// TIA Portal project "TIA_Proiect_Sortare_Cutii" (V15.1)

(* hardware
DEVICE "S7-1200 station_1"  S7-1200 Station
   slot 0: "Rack_0"  S7-1200 Rack  Rack  V1.0
   slot 1: "PLC_1"  CPU 1215C DC/DC/Rly  6ES7 215-1HG40-0XB0  V4.1
   slot 2: "DI 8x24VDC_1"  SM 1221 DI8 x 24VDC  6ES7 221-1BF30-0XB0  V1.0
DEVICE "HMI_1"  TP900 Comfort
   slot 0: "HMI_1"  TP900 Comfort  6AV2 124-0JC01-0AX0  15.1.0.0
   slot 1: "HMI_RT_1"  TP900 Comfort  6AV2 124-0JC01-0AX0  15.1.0.0
   slot 5: "HMI_1.IE_CP_1"  PROFINET Interface  15.0.1.0
      slot 1: "PROFINET Interface_1"  PROFINET Interface
         slot 1: "Port_1"  Port
         slot 2: "Port_2"  Port
   slot 7: "HMI_1.MPI/DP_CP_1"  MPI/DP Interface  15.0.1.0
*)

// ===== PLC "PLC_1"  CPU 1215C DC/DC/Rly =====

VAR_GLOBAL   // PLC tag table "Panel"
   "Running" AT %M20.0 : Bool;
   "Panel_IN" AT %I0.0 : "Equip_panel_IN_t";
   "Panel_QD" AT %Q0.0 : "Equip_panel_QD_t";
   "Panel_counter" AT %QW20 : Int;
END_VAR

VAR_GLOBAL   // PLC tag table "BoxLoad_Sorter"
   "BL_entry_sensor" AT %I1.7 : Bool;
   "BL_sorter_IN" AT %I1.0 : "Equip_sorter_IN_t";
   "BL_sorter_QD" AT %Q1.0 : "Equip_sorter_QD_t";
   "BL_entry_conveyor" AT %Q1.4 : Bool;
   "BL_left_conveyor" AT %Q1.5 : Bool;
   "BL_right_conveyor" AT %Q1.6 : Bool;
END_VAR

VAR_GLOBAL   // PLC tag table "Warehouse1"
   "WH1_entry_crane_IN" AT %I2.0 : "Equip_crane_IN_t";
   "WH1_wait_sensor" AT %I2.5 : Bool;
   "WH1_entry_sensor" AT %I2.6 : Bool;
   "WH1_exit_crane_IN" AT %I3.0 : "Equip_crane_IN_t";
   "WH1_exit_sensor" AT %I3.5 : Bool;
   "WH1_entry_crane_QD" AT %Q2.0 : "Equip_crane_QD_t";
   "WH1_entry_crane_TP" AT %QW22 : Int;
   "WH1_exit_crane_TP" AT %QW24 : Int;
   "WH1_exit_crane_QD" AT %Q3.0 : "Equip_crane_QD_t";
   "WH1_load_conveyor" AT %Q2.3 : Bool;
   "WH1_unload_conveyor" AT %Q3.3 : Bool;
   "WH1_exit_conveyor" AT %Q3.4 : Bool;
   "WH1_exit_curved_conveyor" AT %Q3.5 : Bool;
   "WH1_entry_crane_free" AT %M2.0 : Bool;
END_VAR

VAR_GLOBAL   // PLC tag table "Scale1"
   "Elevator1_IN" AT %I4.0 : "Equip_elevator_IN_t";
   "Elevator1_QD" AT %Q4.0 : "Equip_elevator_QD_t";
   "Scale1_entry_sensor" AT %I4.2 : Bool;
   "Scale1_conveyor_sensor" AT %I4.3 : Bool;
   "Elevator1_free" AT %M4.0 : Bool;
END_VAR

VAR_GLOBAL   // PLC tag table "Clock"
   "Clock_10Hz" AT %M0.0 : Bool;
   "Clock_5Hz" AT %M0.1 : Bool;
   "Clock_2.5Hz" AT %M0.2 : Bool;
   "Clock_2Hz" AT %M0.3 : Bool;
   "Clock_1.25Hz" AT %M0.4 : Bool;
   "Clock_1Hz" AT %M0.5 : Bool;
   "Clock_0.625Hz" AT %M0.6 : Bool;
   "Clock_0.5Hz" AT %M0.7 : Bool;
   "Clock_Byte" AT %MB0 : Byte;
END_VAR

TYPE "Info_RFID_t"
   STRUCT
      Serial_Number : Int;
      Box_Type : Int;
      Exit_DateTime : DTL;
   END_STRUCT;
END_TYPE

TYPE "Obj_box_t"
   STRUCT
      Number : Int;
      "Type" : Int;   // 1 - Small box, 2 - Medium box, 3 - Big box
      Weight : Real;
      State : Int;
   END_STRUCT;
END_TYPE

TYPE "Info_OnTime_t"
   STRUCT
      On_time_secs : Int;
      On_time_mins : Int;
      On_time_hours : Int;
   END_STRUCT;
END_TYPE

TYPE "Equip_RFID_t"
   STRUCT
      IN : Struct
         CommandID : Int;
         Status : Int;
         Read_data : Int;
      END_STRUCT;
      QD : Struct
         Command : Int;
         Execute_command : Bool;
         Memory_index : Int;
         Write_data : Int;
      END_STRUCT;
   END_STRUCT;
END_TYPE

// folder: Crane_t

TYPE "Equip_crane_IN_t"
   STRUCT
      At_left : Bool;
      At_middle : Bool;
      At_right : Bool;
      Moving_X : Bool;
      Moving_Z : Bool;
   END_STRUCT;
END_TYPE

TYPE "Equip_crane_QD_t"
   STRUCT
      Forks_left : Bool;
      Forks_right : Bool;
      Lift : Bool;
   END_STRUCT;
END_TYPE

TYPE "Equip_crane_QW_t"
   STRUCT
      Target_position : Int;
   END_STRUCT;
END_TYPE

// folder: Elevator_t

TYPE "Equip_elevator_IN_t"
   STRUCT
      Left_limit : Bool;
      Right_limit : Bool;
   END_STRUCT;
END_TYPE

TYPE "Equip_elevator_QD_t"
   STRUCT
      Conveyor_fwd : Bool;
      Conveyor_bwd : Bool;
   END_STRUCT;
END_TYPE

TYPE "Equip_elevator_IW_t"
   STRUCT
      Position : Real;
   END_STRUCT;
END_TYPE

TYPE "Equip_elevator_QW_t"
   STRUCT
      Target_position : Real;
   END_STRUCT;
END_TYPE

// folder: Panel_t

TYPE "Equip_panel_IN_t"
   STRUCT
      Start : Bool;
      Stop : Bool;
      Reset : Bool;
      E_stop : Bool;
      Auto : Bool;
      Manual : Bool;
   END_STRUCT;
END_TYPE

TYPE "Equip_panel_QD_t"
   STRUCT
      Start_light : Bool;
      Stop_light : Bool;
      Reset_light : Bool;
   END_STRUCT;
END_TYPE

// folder: Sorter_t

TYPE "Equip_sorter_IN_t"
   STRUCT
      At_left : Bool;
      At_right : Bool;
      Loaded : Bool;
      Pallet : Bool;
      Low : Bool;
      Middle : Bool;
      High : Bool;
   END_STRUCT;
END_TYPE

TYPE "Equip_sorter_QD_t"
   STRUCT
      Chain_left : Bool;
      Chain_right : Bool;
      Load : Bool;
      Unload : Bool;
   END_STRUCT;
END_TYPE

// folder: 01_Box_sorting

DATA_BLOCK "Box_Sorter_DB"   // DB1
{ S7_Optimized_Access := 'TRUE' }
VERSION : 0.1
// stored: InstanceOfName Box_Sorter
"Box_Sorter"
BEGIN
END_DATA_BLOCK

// folder: 03_Warehouse1

DATA_BLOCK "Warehouse1_control_DB"   // DB5
{ S7_Optimized_Access := 'TRUE' }
VERSION : 0.1
// stored: InstanceOfName Warehouse1_control
"Warehouse1_control"
BEGIN
END_DATA_BLOCK

// folder: Logistics

DATA_BLOCK "Global_data"   // DB2
{ S7_Optimized_Access := 'TRUE' }
VERSION : 0.1
   VAR
      State_sorting : Int := 1;
      Box_object : Array[1..1000] of "Obj_box_t";
      Box_count : Int;
      Box_current : "Obj_box_t";
      State_W1_EntryCrane : Int;
      State_W1_ExitCrane : Int;
      WH1_entry_crane : "Equip_crane_IN_t";
   END_VAR
BEGIN
END_DATA_BLOCK

DATA_BLOCK "Warehouse1"   // DB3
{ S7_Optimized_Access := 'TRUE' }
VERSION : 0.1
   VAR
      Store_count : Array[1..54] of Int;
      Free_positions : Int;
      Occupied_positions : Int;
   END_VAR
BEGIN
END_DATA_BLOCK

DATA_BLOCK "HMI"   // DB4
{ S7_Optimized_Access := 'TRUE' }
VERSION : 0.1
   VAR
      START_CMD : Struct
         BL_sorting : Struct
            BL_entry_conveyor : Bool;
            BL_load_sort : Bool;
            BL_unload_sort : Bool;
            BL_transf_left : Bool;
            BL_transf_right : Bool;
            BL_left_conveyor : Bool;
            BL_right_conveyor : Bool;
         END_STRUCT;
         Warehouse1 : Struct
            WH1_load_conveyor : Bool;
            Entry_crane : Struct
               Target_position : Int;
               Forks_left : Bool;
               Forks_right : Bool;
               Lift : Bool;
            END_STRUCT;
            Exit_crane : Struct
               Target_position : Int;
               Forks_left : Bool;
               Forks_right : Bool;
               Lift : Bool;
            END_STRUCT;
         END_STRUCT;
         Elevator1 : Struct
            Elevator1_fwd : Bool;
            Elevator1_bwd : Bool;
         END_STRUCT;
         Elevator2 : Struct
            Elevator2_fwd : Bool;
            Elevator2_bwd : Bool;
         END_STRUCT;
         Weight_scale : Struct
            Scale_conveyor_fwd : Bool;
            Scale_conveyor_bwd : Bool;
         END_STRUCT;
      END_STRUCT;
      STOP_CMD : Struct
         BL_sorting : Struct
            BL_entry_conveyor : Bool;
            BL_load_sort : Bool;
            BL_unload_sort : Bool;
            BL_transf_left : Bool;
            BL_transf_right : Bool;
            BL_left_conveyor : Bool;
            BL_right_conveyor : Bool;
         END_STRUCT;
         Warehouse1 : Struct
            WH1_load_conveyor : Bool;
            Entry_crane : Struct
               Target_position : Int;
               Forks_left : Bool;
               Forks_right : Bool;
               Lift : Bool;
            END_STRUCT;
            Exit_crane : Struct
               Target_position : Int;
               Forks_left : Bool;
               Forks_right : Bool;
               Lift : Bool;
            END_STRUCT;
         END_STRUCT;
         Elevator1 : Struct
            Elevator1_fwd : Bool;
            Elevator1_bwd : Bool;
         END_STRUCT;
         Elevator2 : Struct
            Elevator2_fwd : Bool;
            Elevator2_bwd : Bool;
         END_STRUCT;
         Weight_scale : Struct
            Scale_conveyor_fwd : Bool;
            Scale_conveyor_bwd : Bool;
         END_STRUCT;
      END_STRUCT;
      MAN_CTRL : Struct
         BL_sorting : Struct
            BL_entry_conveyor : Bool;
            BL_load_sort : Bool;
            BL_unload_sort : Bool;
            BL_transf_left : Bool;
            BL_transf_right : Bool;
            BL_left_conveyor : Bool;
            BL_right_conveyor : Bool;
         END_STRUCT;
         Warehouse1 : Struct
            WH1_load_conveyor : Bool;
            Entry_crane : Struct
               Target_position : Int;
               Forks_left : Bool;
               Forks_right : Bool;
               Lift : Bool;
            END_STRUCT;
            Exit_crane : Struct
               Target_position : Int;
               Forks_left : Bool;
               Forks_right : Bool;
               Lift : Bool;
            END_STRUCT;
         END_STRUCT;
         Elevator1 : Struct
            Elevator1_fwd : Bool;
            Elevator1_bwd : Bool;
         END_STRUCT;
         Elevator2 : Struct
            Elevator2_fwd : Bool;
            Elevator2_bwd : Bool;
         END_STRUCT;
         Weight_scale : Struct
            Scale_conveyor_fwd : Bool;
            Scale_conveyor_bwd : Bool;
         END_STRUCT;
      END_STRUCT;
   END_VAR
BEGIN
END_DATA_BLOCK

// folder: (top level)

FUNCTION "Manual_control" : Void   // FC4, SCL
{ S7_Optimized_Access := 'TRUE' }
VERSION : 0.1
BEGIN
   IF ("Panel_IN".Manual) THEN

       REGION CONVEYOR_MANUAL_CONTROL

           REGION BOX_LOAD_SORTING_CONVEYOR_CONTROL
               //--------- BOX LOAD ENTRY CONVEYOR
               IF ("HMI".START_CMD.BL_sorting.BL_entry_conveyor) THEN
                   "HMI".MAN_CTRL.BL_sorting.BL_entry_conveyor := TRUE;
               ELSE
                   "HMI".MAN_CTRL.BL_sorting.BL_entry_conveyor := FALSE;
               END_IF;

               //!!!!!!!!!!!!!!!!!!!!!!!!!!!!!!!!!
               // ADD HMI STOP FOR EACH EQUIPMENT
               //!!!!!!!!!!!!!!!!!!!!!!!!!!!!!!!!!
               //
               //--------- BOX LOAD SORT CONVEYOR 
               IF ("HMI".START_CMD.BL_sorting.BL_load_sort) THEN
                   "HMI".MAN_CTRL.BL_sorting.BL_load_sort := TRUE;
                   "HMI".MAN_CTRL.BL_sorting.BL_unload_sort := FALSE;
               ELSE
                   "HMI".MAN_CTRL.BL_sorting.BL_load_sort := FALSE;
               END_IF;

               IF ("HMI".START_CMD.BL_sorting.BL_unload_sort) THEN
                   "HMI".MAN_CTRL.BL_sorting.BL_unload_sort := TRUE;
                   "HMI".MAN_CTRL.BL_sorting.BL_load_sort := FALSE;
               ELSE
                   "HMI".MAN_CTRL.BL_sorting.BL_unload_sort := FALSE;
               END_IF;

               IF ("HMI".START_CMD.BL_sorting.BL_transf_left) THEN
                   "HMI".MAN_CTRL.BL_sorting.BL_transf_left := TRUE;
                   "HMI".MAN_CTRL.BL_sorting.BL_transf_right := FALSE;
               ELSE
                   "HMI".MAN_CTRL.BL_sorting.BL_transf_left := FALSE;
               END_IF;

               IF ("HMI".START_CMD.BL_sorting.BL_transf_right) THEN
                   "HMI".MAN_CTRL.BL_sorting.BL_transf_right := TRUE;
                   "HMI".MAN_CTRL.BL_sorting.BL_transf_left := FALSE;
               ELSE
                   "HMI".MAN_CTRL.BL_sorting.BL_transf_right := FALSE;
               END_IF;
           END_REGION

           //--------- WAREHOUSE 1 ENTRY CONVEYOR
           IF ("HMI".START_CMD.BL_sorting.BL_right_conveyor) THEN
               "HMI".MAN_CTRL.BL_sorting.BL_right_conveyor := TRUE;
           ELSE
               "HMI".MAN_CTRL.BL_sorting.BL_right_conveyor := FALSE;
           END_IF;

           //--------- ELEVATOR 1 ENTRY CONVEYOR
           IF ("HMI".START_CMD.BL_sorting.BL_left_conveyor) THEN
               "HMI".MAN_CTRL.BL_sorting.BL_left_conveyor := TRUE;
           ELSE
               "HMI".MAN_CTRL.BL_sorting.BL_left_conveyor := FALSE;
           END_IF;

           REGION ELEVATOR1_CONVEYOR_CONTROL
               IF ("HMI".START_CMD.Elevator1.Elevator1_fwd) THEN
                   "HMI".MAN_CTRL.Elevator1.Elevator1_fwd := TRUE;
                   "HMI".MAN_CTRL.Elevator1.Elevator1_bwd := FALSE;
               ELSE
                   "HMI".MAN_CTRL.Elevator1.Elevator1_fwd := FALSE;
               END_IF;

               IF ("HMI".START_CMD.Elevator1.Elevator1_fwd) THEN
                   "HMI".MAN_CTRL.Elevator1.Elevator1_bwd := TRUE;
                   "HMI".MAN_CTRL.Elevator1.Elevator1_fwd := FALSE;
               ELSE
                   "HMI".MAN_CTRL.Elevator1.Elevator1_bwd := FALSE;
               END_IF;
           END_REGION

       END_REGION 

       REGION CRANE_MANUAL_CONTROL

       END_REGION 

   END_IF;
END_FUNCTION

FUNCTION "MHJ-PLC-Lab-Function-S71200" : Void   // FC9000, SCL
{ S7_Optimized_Access := 'TRUE' }
VERSION : 0.1
   VAR_TEMP
      rdTimeReturn : Int;
      outputTime : DTL;
      SyncVal : Byte;
      forVal : Int;
      forVal_2 : Int;
      Value : Byte;
   END_VAR
   VAR CONSTANT
      CompVal : Byte := 16#34;
      Value_01 : Byte := 16#11;
      Value_01_DW : DWord := 16#A165_D992;
      Value_02_DW : DWord := 16#58BE_4401;
   END_VAR
BEGIN

   #Value:=PEEK(area := 16#82,
        dbNumber := 0,
        byteOffset := 511);
   #Value := #Value + 1;

   POKE(area := 16#82,
        dbNumber := 0,
        byteOffset := 511,
        value := #Value);

   POKE(area:=16#81,
        dbNumber:=0,
        byteOffset:=1016,
        value:=#Value_01_DW);
   POKE(area := 16#81,
        dbNumber := 0,
        byteOffset := 1020,
        value := #Value_02_DW);

   POKE(area := 16#81,
        dbNumber := 0,
        byteOffset := 511,
        value := B#16#00);

   FOR #forVal := 0 TO 120 DO
       FOR #forVal_2:=0 TO 10 DO
           #rdTimeReturn:=RD_SYS_T(#outputTime);
           #rdTimeReturn := WR_SYS_T(#outputTime);
           #rdTimeReturn := RD_SYS_T(#outputTime);
           #rdTimeReturn := WR_SYS_T(#outputTime);
       END_FOR;
       #SyncVal:= PEEK(area := 16#81,
                      dbNumber := 0,
                      byteOffset := 511);
       IF #SyncVal = #CompVal THEN
          GOTO M_1;
       END_IF;
   END_FOR;
   RETURN;

   M_1:
   POKE(area := 16#81,
        dbNumber := 0,
        byteOffset := 511,
        value := B#16#0);
END_FUNCTION

ORGANIZATION_BLOCK "Main"   // OB1, LAD, ProgramCycle
TITLE = "Main Program Sweep (Cycle)"
{ S7_Optimized_Access := 'TRUE' }
VERSION : 0.1
   VAR_INPUT
      Initial_Call : Bool;   // Initial call of this OB
      Remanence : Bool;   // =True, if remanent data are available
   END_VAR
BEGIN

REGION Network 1: FactoryIO connection
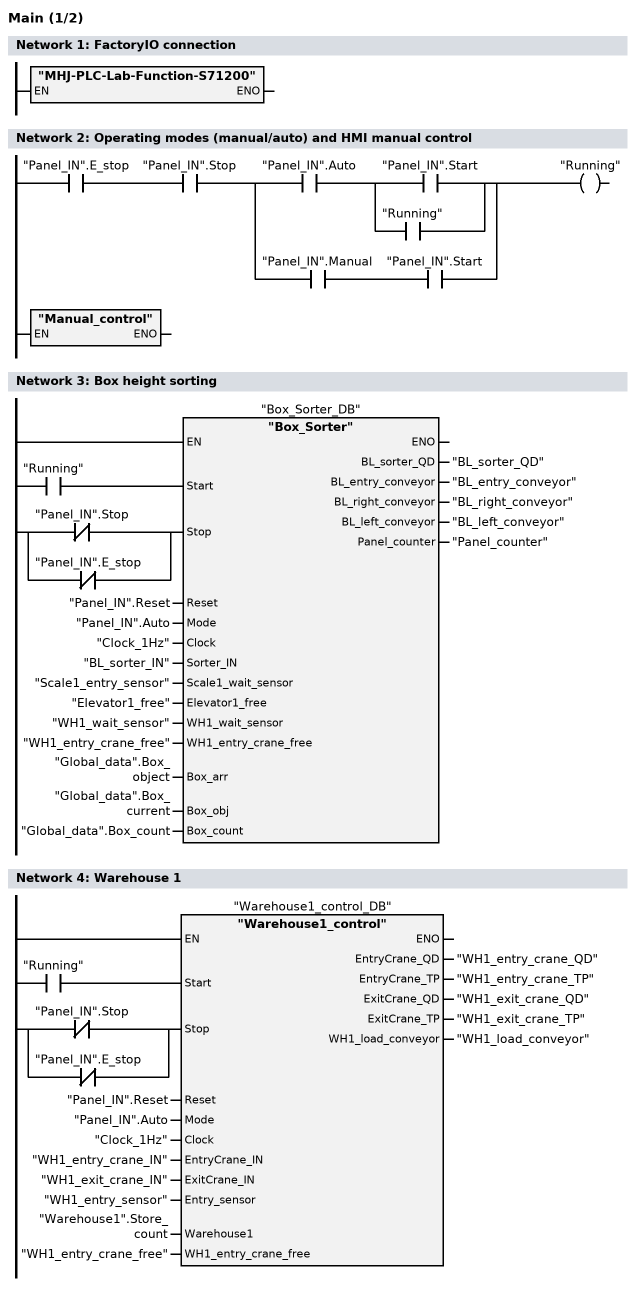
   RUNG wire#powerrail
      "MHJ-PLC-Lab-Function-S71200"()
   END_RUNG
   // the same network as SCL:
   "MHJ-PLC-Lab-Function-S71200"();
END_REGION

REGION Network 2: Operating modes (manual/auto) and HMI manual control
   RUNG wire#powerrail
      Contact( "Panel_IN".E_stop )
      Contact( "Panel_IN".Stop )
      wire#w1
      Contact( "Panel_IN".Auto )
      wire#w2
      Contact( "Panel_IN".Start )
      wire#w3
      Coil( "Running" )
   END_RUNG
   RUNG wire#w2
      Contact( "Running" )
   END_RUNG wire#w3
   RUNG wire#w1
      Contact( "Panel_IN".Manual )
      Contact( "Panel_IN".Start )
   END_RUNG wire#w3
   RUNG wire#powerrail
      "Manual_control"()
   END_RUNG
   // the same network as SCL:
   "Running" := "Panel_IN".E_stop AND "Panel_IN".Stop AND (("Panel_IN".Auto AND ("Panel_IN".Start OR "Running")) OR ("Panel_IN".Manual AND "Panel_IN".Start));
   "Manual_control"();
END_REGION

REGION Network 3: Box height sorting
   RUNG wire#powerrail
      "Box_Sorter_DB"(Start := wire#w1, Stop := wire#w2, Reset := "Panel_IN".Reset, Mode := "Panel_IN".Auto, Clock := "Clock_1Hz", Sorter_IN := "BL_sorter_IN", Scale1_wait_sensor := "Scale1_entry_sensor", Elevator1_free := "Elevator1_free", WH1_wait_sensor := "WH1_wait_sensor", WH1_entry_crane_free := "WH1_entry_crane_free", Box_arr := "Global_data".Box_object, Box_obj := "Global_data".Box_current, Box_count := "Global_data".Box_count, BL_sorter_QD => "BL_sorter_QD", BL_entry_conveyor => "BL_entry_conveyor", BL_right_conveyor => "BL_right_conveyor", BL_left_conveyor => "BL_left_conveyor", Panel_counter => "Panel_counter")
   END_RUNG
   RUNG wire#powerrail
      Contact( "Running" )
   END_RUNG wire#w1
   RUNG wire#powerrail
      I_Contact( "Panel_IN".Stop )
   END_RUNG wire#w2
   RUNG wire#powerrail
      I_Contact( "Panel_IN".E_stop )
   END_RUNG wire#w2
   // the same network as SCL:
   "Box_Sorter_DB"(Start := "Running",   // "Box_Sorter"
                   Stop := NOT "Panel_IN".Stop OR NOT "Panel_IN".E_stop,
                   Reset := "Panel_IN".Reset,
                   Mode := "Panel_IN".Auto,
                   Clock := "Clock_1Hz",
                   Sorter_IN := "BL_sorter_IN",
                   Scale1_wait_sensor := "Scale1_entry_sensor",
                   Elevator1_free := "Elevator1_free",
                   WH1_wait_sensor := "WH1_wait_sensor",
                   WH1_entry_crane_free := "WH1_entry_crane_free",
                   Box_arr := "Global_data".Box_object,
                   Box_obj := "Global_data".Box_current,
                   Box_count := "Global_data".Box_count,
                   BL_sorter_QD => "BL_sorter_QD",
                   BL_entry_conveyor => "BL_entry_conveyor",
                   BL_right_conveyor => "BL_right_conveyor",
                   BL_left_conveyor => "BL_left_conveyor",
                   Panel_counter => "Panel_counter");
END_REGION

REGION Network 4: Warehouse 1
   RUNG wire#powerrail
      "Warehouse1_control_DB"(Start := wire#w1, Stop := wire#w2, Reset := "Panel_IN".Reset, Mode := "Panel_IN".Auto, Clock := "Clock_1Hz", EntryCrane_IN := "WH1_entry_crane_IN", ExitCrane_IN := "WH1_exit_crane_IN", Entry_sensor := "WH1_entry_sensor", Warehouse1 := "Warehouse1".Store_count, WH1_entry_crane_free := "WH1_entry_crane_free", EntryCrane_QD => "WH1_entry_crane_QD", EntryCrane_TP => "WH1_entry_crane_TP", ExitCrane_QD => "WH1_exit_crane_QD", ExitCrane_TP => "WH1_exit_crane_TP", WH1_load_conveyor => "WH1_load_conveyor")
   END_RUNG
   RUNG wire#powerrail
      Contact( "Running" )
   END_RUNG wire#w1
   RUNG wire#powerrail
      I_Contact( "Panel_IN".Stop )
   END_RUNG wire#w2
   RUNG wire#powerrail
      I_Contact( "Panel_IN".E_stop )
   END_RUNG wire#w2
   // the same network as SCL:
   "Warehouse1_control_DB"(Start := "Running",   // "Warehouse1_control"
                           Stop := NOT "Panel_IN".Stop OR NOT "Panel_IN".E_stop,
                           Reset := "Panel_IN".Reset,
                           Mode := "Panel_IN".Auto,
                           Clock := "Clock_1Hz",
                           EntryCrane_IN := "WH1_entry_crane_IN",
                           ExitCrane_IN := "WH1_exit_crane_IN",
                           Entry_sensor := "WH1_entry_sensor",
                           Warehouse1 := "Warehouse1".Store_count,
                           WH1_entry_crane_free := "WH1_entry_crane_free",
                           EntryCrane_QD => "WH1_entry_crane_QD",
                           EntryCrane_TP => "WH1_entry_crane_TP",
                           ExitCrane_QD => "WH1_exit_crane_QD",
                           ExitCrane_TP => "WH1_exit_crane_TP",
                           WH1_load_conveyor => "WH1_load_conveyor");
END_REGION

REGION Network 5: Button lights
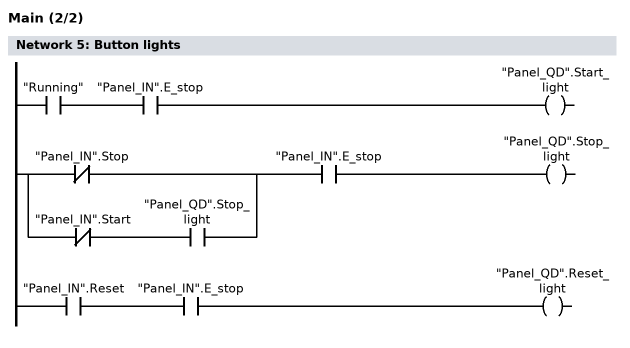
   RUNG wire#powerrail
      Contact( "Running" )
      Contact( "Panel_IN".E_stop )
      Coil( "Panel_QD".Start_light )
   END_RUNG
   RUNG wire#powerrail
      I_Contact( "Panel_IN".Stop )
      wire#w1
      Contact( "Panel_IN".E_stop )
      Coil( "Panel_QD".Stop_light )
   END_RUNG
   RUNG wire#powerrail
      I_Contact( "Panel_IN".Start )
      Contact( "Panel_QD".Stop_light )
   END_RUNG wire#w1
   RUNG wire#powerrail
      Contact( "Panel_IN".Reset )
      Contact( "Panel_IN".E_stop )
      Coil( "Panel_QD".Reset_light )
   END_RUNG
   // the same network as SCL:
   "Panel_QD".Start_light := "Running" AND "Panel_IN".E_stop;
   "Panel_QD".Stop_light := (NOT "Panel_IN".Stop OR (NOT "Panel_IN".Start AND "Panel_QD".Stop_light)) AND "Panel_IN".E_stop;
   "Panel_QD".Reset_light := "Panel_IN".Reset AND "Panel_IN".E_stop;
END_REGION
END_ORGANIZATION_BLOCK

// folder: 00_Conveyor

FUNCTION_BLOCK "Sort_conveyor_control"   // FB5, SCL
{ S7_Optimized_Access := 'TRUE' }
VERSION : 0.1
   VAR_INPUT
      Start : Bool;
      Stop : Bool;
      Reset : Bool;
      Mode : Bool;   // Using Auto for input 0-MAN 1-AUTO
      Clock : Bool;
      TR_left : Bool;
      TR_right : Bool;
      P_load : Bool;
      P_unload : Bool;
   END_VAR
   VAR_OUTPUT
      Chain_left : Bool;
      Chain_right : Bool;
      Load : Bool;
      Unload : Bool;
   END_VAR
   VAR
      Status : Int;
      Equipment_time_counter_Instance : "Equipment_time_counter";
      On_time : "Info_OnTime_t";
   END_VAR
   VAR CONSTANT
      On : Int := 5;
      Off : Int := 1;
      No_data : Int := 0;
      MAN : Bool := 0;
      AUTO : Bool := 1;
   END_VAR
BEGIN

   IF (#Mode = #MAN) THEN
       "Manual_control"();
   END_IF;

   IF (#Mode = #AUTO) THEN
       IF (#Start) THEN
           IF (#P_load) THEN
               #Load := TRUE;
               #Unload := FALSE;
           ELSE
               #Load := FALSE;
           END_IF;

           IF (#P_unload) THEN
               #Unload := TRUE;
               #Load := FALSE;
           ELSE
               #Unload := FALSE;
           END_IF;

           IF (#TR_left) THEN
               #Chain_left := TRUE;
               #Chain_right := FALSE;
           ELSE
               #Chain_left := FALSE;
           END_IF;

           IF (#TR_right) THEN
               #Chain_right := TRUE;
               #Chain_left := FALSE;
           ELSE
               #Chain_right := FALSE;
           END_IF;
       ELSIF #Stop THEN
           #Chain_left := FALSE;
           #Chain_right := FALSE;
           #Load := FALSE;
           #Unload := FALSE;
       END_IF;
   END_IF;

   IF (#Reset) THEN
       #On_time.On_time_hours := 0;
       #On_time.On_time_mins := 0;
       #On_time.On_time_secs := 0;
       #Chain_left := FALSE;
       #Chain_right := FALSE;
       #Load := FALSE;
       #Unload := FALSE;
       #Status := #Off;
   END_IF;

   IF (#Load OR #Unload OR #Chain_left OR #Chain_right) THEN
       #Equipment_time_counter_Instance(Clock := #Clock,
                                        On_time := #On_time);

       #Status := #On;
   ELSE
       #Status := #Off;
   END_IF;
END_FUNCTION_BLOCK

FUNCTION_BLOCK "Conveyor_control"   // FB8, SCL
{ S7_Optimized_Access := 'TRUE' }
VERSION : 0.1
   VAR_INPUT
      Start : Bool;
      Stop : Bool;
      Reset : Bool;
      Mode : Bool;   // Using Auto for input 0-MAN 1-AUTO
      Clock : Bool;
      Fwd : Bool;
      Bwd : Bool;
   END_VAR
   VAR_OUTPUT
      Conveyor_fwd : Bool;
      Conveyor_bwd : Bool;
   END_VAR
   VAR
      Status : Int;
      Equipment_time_counter_Instance : "Equipment_time_counter";
      On_time : "Info_OnTime_t";
   END_VAR
   VAR CONSTANT
      On : Int := 5;
      Off : Int := 1;
      No_data : Int := 0;
      MAN : Bool := 0;
      AUTO : Bool := 1;
   END_VAR
BEGIN

   IF (#Mode = #MAN) THEN
       "Manual_control"();
   END_IF;

   IF (#Mode = #AUTO) THEN
       IF (#Start) THEN
           IF (#Fwd) THEN
               #Conveyor_fwd := TRUE;
               #Conveyor_bwd := FALSE;
           ELSE
               #Conveyor_fwd := FALSE;
           END_IF;

           IF (#Bwd) THEN
               #Conveyor_bwd := TRUE;
               #Conveyor_fwd := FALSE;
           ELSE
               #Conveyor_bwd := FALSE;
           END_IF;
       ELSIF (#Stop) THEN
           #Conveyor_fwd := FALSE;
           #Conveyor_bwd := FALSE;
       END_IF;
   END_IF;

   IF (#Reset) THEN
       #On_time.On_time_hours := 0;
       #On_time.On_time_mins := 0;
       #On_time.On_time_secs := 0;
       #Conveyor_fwd := FALSE;
       #Status := #Off;
   END_IF;

   IF (#Conveyor_fwd OR #Conveyor_fwd) THEN
       #Equipment_time_counter_Instance(Clock:=#Clock,
                                        On_time:=#On_time);

       #Status := #On;
   ELSE
       #Status := #Off;
   END_IF;
END_FUNCTION_BLOCK

// folder: 01_Box_sorting

FUNCTION_BLOCK "Box_Sorter"   // FB2, SCL
{ S7_Optimized_Access := 'TRUE' }
VERSION : 0.1
   VAR_INPUT
      Start : Bool;
      Stop : Bool;
      Reset : Bool;
      Mode : Bool;   // Using Auto for input 0-MAN 1-AUTO
      Clock : Bool;
      Sorter_IN : "Equip_sorter_IN_t";
      Scale1_wait_sensor : Bool;
      Elevator1_free : Bool;   // 0 - Elevator in use, 1 - Elevator free
      WH1_wait_sensor : Bool;
      WH1_entry_crane_free : Bool;   // 0 - Crane in use, 1 - Crane free
   END_VAR
   VAR_OUTPUT
      BL_sorter_QD : "Equip_sorter_QD_t";
      BL_entry_conveyor : Bool;
      BL_right_conveyor : Bool;
      BL_left_conveyor : Bool;
      Panel_counter : Int;
   END_VAR
   VAR_IN_OUT
      Box_arr : Array[1..1000] of "Obj_box_t";
      Box_obj : "Obj_box_t";
      Box_count : Int;
   END_VAR
   VAR
      Pallet_detected : Bool;
      Pallet_loaded : Bool;
      Pallet_transfer_left : Bool;
      Pallet_transfer_right : Bool;
      Pallet_at_left : Bool;
      Pallet_at_right : Bool;
      State : Int := 1;
      On_time : "Info_OnTime_t";
      BL_entry_conveyor_FB : "Conveyor_control";
      BL_sort_conveyor_FB : "Sort_conveyor_control";
      BL_right_conveyor_FB : "Conveyor_control";
      WH1_load_conveyor_FB : "Conveyor_control";
      BL_left_conveyor_FB : "Conveyor_control";
      TR_left_sensor_FB : "Sensor_control";
      TR_right_sensor_FB : "Sensor_control";
      Load_sensor_FB : "Sensor_control";
      Pallet_sensor_FB : "Sensor_control";
      Low_sensor_FB : "Sensor_control";
      Middle_sensor_FB : "Sensor_control";
      High_sensor_FB : "Sensor_control";
      Timer_check_stuck : TON_TIME;
      Timer_check_missing : TON_TIME;
      Elevator1_conveyor_FB : "Conveyor_control";
      WH1_wait_sensor_FB : "Sensor_control";
      Scale1_wait_sensor_FB : "Sensor_control";
   END_VAR
   VAR CONSTANT
      MAN : Bool := 0;
      AUTO : Bool := 1;
      PalletToSorter : Int := 1;
      PalletTransferLR : Int := 2;
      SmallBox : Int := 1;
      MedBox : Int := 2;
      LargeBox : Int := 3;
   END_VAR
BEGIN

   REGION FB_calls_for_equipment_and_sensors
       REGION ACTUATORS
           #BL_entry_conveyor_FB(Start := #Start,
                                 Stop := #Stop,
                                 Reset := #Reset,
                                 Mode := #Mode,
                                 Clock := #Clock,
                                 Fwd := ("HMI".MAN_CTRL.BL_sorting.BL_entry_conveyor)
                                 OR (#State = #PalletToSorter AND NOT #Pallet_loaded)
                                 OR (#State <> #PalletToSorter AND NOT #Pallet_detected),
                                 Bwd := FALSE,
                                 Conveyor_fwd => #BL_entry_conveyor);

           #BL_sort_conveyor_FB(Start := #Start,
                                Stop := #Stop,
                                Reset := #Reset,
                                Mode := #Mode,
                                Clock := #Clock,
                                TR_left := ("HMI".MAN_CTRL.BL_sorting.BL_transf_left) //CHANGE TO DEPEND ON IF CONVEYOR IS RUNNING
                                OR (#State <> #PalletToSorter AND #Pallet_transfer_left),
                                TR_right := ("HMI".MAN_CTRL.BL_sorting.BL_transf_right)
                                OR (#State <> #PalletToSorter AND #Pallet_transfer_right),
                                P_load := ("HMI".MAN_CTRL.BL_sorting.BL_load_sort)
                                OR (#State = #PalletToSorter AND NOT #Pallet_loaded),
                                P_unload := ("HMI".MAN_CTRL.BL_sorting.BL_unload_sort),
                                Chain_left => #BL_sorter_QD.Chain_left,
                                Chain_right => #BL_sorter_QD.Chain_right,
                                Load => #BL_sorter_QD.Load,
                                Unload => #BL_sorter_QD.Unload);

           #BL_right_conveyor_FB(Start := #Start,
                                 Stop := #Stop,
                                 Reset := #Reset,
                                 Mode := #Mode,
                                 Clock := #Clock,
                                 Fwd := ("HMI".MAN_CTRL.BL_sorting.BL_right_conveyor)
                                 OR (#WH1_entry_crane_free OR NOT #Pallet_at_right),
                                 Bwd := FALSE,
                                 Conveyor_fwd => #BL_right_conveyor);

           #BL_left_conveyor_FB(Start := #Start,
                                Stop := #Stop,
                                Reset := #Reset,
                                Mode := #Mode,
                                Clock := #Clock,
                                Fwd := ("HMI".MAN_CTRL.BL_sorting.BL_left_conveyor)
                                OR (#Elevator1_free OR NOT #Pallet_at_left),
                                Bwd := FALSE,
                                Conveyor_fwd => #BL_left_conveyor);

       END_REGION

       REGION SENSORS
           #Load_sensor_FB(Sensor := #Sorter_IN.Loaded,
                           Debounce_time := T#200ms,
                           Timeout := T#2000ms,
                           Enabled := TRUE);

           #Pallet_sensor_FB(Sensor := #Sorter_IN.Pallet,
                             Debounce_time := T#100ms,
                             Timeout := T#2000ms,
                             Enabled := TRUE);

           #Low_sensor_FB(Sensor := #Sorter_IN.Low,
                          Debounce_time := T#200ms,
                          Timeout := T#2000ms,
                          Enabled := TRUE);

           #Middle_sensor_FB(Sensor := #Sorter_IN.Middle,
                             Debounce_time := T#200ms,
                             Timeout := T#2000ms,
                             Enabled := TRUE);

           #High_sensor_FB(Sensor := #Sorter_IN.High,
                           Debounce_time := T#200ms,
                           Timeout := T#2000ms,
                           Enabled := TRUE);

           #TR_left_sensor_FB(Sensor := #Sorter_IN.At_left,
                              Debounce_time := T#200ms,
                              Timeout := T#2000ms,
                              Enabled := TRUE);

           #TR_right_sensor_FB(Sensor := #Sorter_IN.At_right,
                               Debounce_time := T#200ms,
                               Timeout := T#2000ms,
                               Enabled := TRUE);

           #Scale1_wait_sensor_FB(Sensor:=#Scale1_wait_sensor,
                                  Debounce_time:=T#100ms,
                                  Timeout:=T#2000ms,
                                  Enabled:=TRUE);

           #WH1_wait_sensor_FB(Sensor:=#WH1_wait_sensor,
                                Debounce_time:=T#100ms,
                                Timeout:=T#2000ms,
                                Enabled:=TRUE);

       END_REGION
   END_REGION

   IF (#Reset) THEN
       #Box_count := 0;
       #State := #PalletToSorter;
   END_IF;

   IF (#Mode = #AUTO) AND (#Start) THEN

       #Panel_counter := #Box_count;

       IF (#Pallet_sensor_FB.Is_busy) THEN
           #Pallet_detected := TRUE;
       ELSE
           #Pallet_detected := FALSE;
       END_IF;

       IF (#Scale1_wait_sensor_FB.Is_free) THEN
           #Pallet_at_left := TRUE;
       ELSE
           #Pallet_at_left := FALSE;
       END_IF;

       IF (#WH1_wait_sensor_FB.Is_free) THEN
           #Pallet_at_right := TRUE;
       ELSE
           #Pallet_at_right := FALSE;
       END_IF;

       CASE #State OF
           #PalletToSorter:  // Step 1, pallet advances to sorter
               REGION Box_type_detection
                   IF (#Pallet_sensor_FB.Is_busy) THEN
                       IF (#Low_sensor_FB.Is_busy) THEN
                           #Box_obj.Type := #SmallBox;
                           IF (#Middle_sensor_FB.Is_busy) THEN
                               #Box_obj.Type := #MedBox;
                               IF (#High_sensor_FB.Is_busy) THEN
                                   #Box_obj.Type := #LargeBox;
                               END_IF;
                           END_IF;
                       END_IF;
                   END_IF;
               END_REGION 

               IF (#Load_sensor_FB.Is_busy) THEN
                   #Pallet_loaded := TRUE;
                   #State := #PalletTransferLR;
                   #Box_count := #Box_count + 1;
               ELSE
                   #Pallet_loaded := FALSE;
               END_IF;

           #PalletTransferLR:  // Step 2, transfer depending on size
               IF ((#Box_obj.Type = #SmallBox) OR (#Box_obj.Type = #MedBox)) THEN
                   IF (NOT #Pallet_at_left) THEN // Schimb sa nu depinda de senzorul de capat
                       #Pallet_transfer_left := TRUE; // ci de o conditie setata de celula cealalta
                       #Pallet_transfer_right := FALSE; // SAU SCHIMB SA DEPINDA DE CONVEIOARELE
                   ELSE                                 // LEFT / RIGHT??
                       #Pallet_transfer_left := FALSE;
                   END_IF;

                   IF (#Pallet_transfer_left AND #TR_left_sensor_FB.R_edge) THEN
                       #Pallet_transfer_left := FALSE;
                       #State := #PalletToSorter;
                   END_IF;
               ELSIF (#Box_obj.Type = #LargeBox) THEN
                   IF (NOT #Pallet_at_right) THEN
                       #Pallet_transfer_left := FALSE;
                       #Pallet_transfer_right := TRUE;
                   ELSE
                       #Pallet_transfer_right := FALSE;
                   END_IF;

                   IF (#Pallet_transfer_right AND #TR_right_sensor_FB.R_edge) THEN
                       #Pallet_transfer_right := FALSE;
                       #State := #PalletToSorter;
                   END_IF;
               ELSE
                   #Pallet_transfer_left := FALSE;
                   #Pallet_transfer_right := FALSE;
               END_IF;

               REGION Check_if_box_stuck_during_transfer
                   IF (#Pallet_transfer_left AND NOT #TR_left_sensor_FB.R_edge) OR
                       (#Pallet_transfer_right AND NOT #TR_right_sensor_FB.R_edge) THEN

                       #Timer_check_stuck(IN := (#Load_sensor_FB.Is_busy),
                                          PT := T#8s);

                       #Timer_check_missing(IN:=(#Load_sensor_FB.Is_free),
                                            PT:=T#8s);

                       IF (#Timer_check_stuck.Q) THEN
                           #Pallet_transfer_left := FALSE;
                           #Pallet_transfer_right := FALSE; // AND ALARM PALLET IS STUCK ON LOADER
                       END_IF;

                       IF (#Timer_check_missing.Q) THEN
                           #Pallet_transfer_left := FALSE;
                           #Pallet_transfer_right := FALSE; // AND ALARM PALLET IS MISSING FROM LOADER
                           #State := #PalletToSorter; // ALSO RESET TO STATE 1
                       END_IF;
                   END_IF;
               END_REGION

           ELSE
               #State := #PalletToSorter;
       END_CASE;

   END_IF;
END_FUNCTION_BLOCK

// folder: 02_Crane_control

FUNCTION_BLOCK "Crane_control"   // FB1, SCL
{ S7_Optimized_Access := 'TRUE' }
VERSION : 0.1
   VAR_INPUT
      Start : Bool;
      Stop : Bool;
      Reset : Bool;
      Mode : Bool;
      Clock : Bool;
      Forks_mLeft : Bool;
      Forks_mRight : Bool;
      Lift : Bool;
      Crane_IN : "Equip_crane_IN_t";
      Setpoint : Int;
   END_VAR
   VAR_OUTPUT
      Crane_QD : "Equip_crane_QD_t";
      Crane_target_position : Int;
   END_VAR
   VAR
      Crane_status : Int;
      Lift_status : Int;
      Equipment_status : Int;
      On_time : "Info_OnTime_t";
      Equipment_time_counter_Instance : "Equipment_time_counter";
      Check_forksL_move : TON_TIME;
      Check_forksR_move : TON_TIME;
      Check_forksM_move : TON_TIME;
      Check_lift_moving : TON_TIME;
      Check_stacker_moving : TON_TIME;
      Check_stacker_stuck : TON_TIME;
      Check_lift_stuck : TON_TIME;
   END_VAR
   VAR CONSTANT
      On : Int := 0;
      Off : Int := 1;
      Moving : Int := 2;
      Stopped : Int := 3;
      LiftStopped : Int := 0;
      LiftMoving : Int := 1;
      MAN : Bool := 0;
      AUTO : Bool := 1;
      Depositing : Bool := 0;
      Extracting : Bool := 1;
      MAX_SETPOINT : Int := 54;
   END_VAR
BEGIN

   IF (#Mode = #MAN) THEN
       "Manual_control"();
   END_IF;

   IF (#Mode = #AUTO) THEN
       IF (#Start) THEN
           IF (#Forks_mLeft) THEN
               #Crane_QD.Forks_left := TRUE;
               #Crane_QD.Forks_right := FALSE;
           ELSE
               #Crane_QD.Forks_left := FALSE;
           END_IF;

           IF (#Forks_mRight) THEN
               #Crane_QD.Forks_left := FALSE;
               #Crane_QD.Forks_right := TRUE;
           ELSE
               #Crane_QD.Forks_right := FALSE;
           END_IF;

           (*IF (#Lift AND #Lift_status = #LiftStopped AND #Crane_status = #Stopped) THEN
               #Crane_QD.Lift := TRUE;
               #Lift_status := #LiftMoving;
           END_IF;

           IF (NOT #Lift AND #Lift_status = #LiftStopped AND #Crane_status = #Stopped) THEN
               #Crane_QD.Lift := FALSE;
               #Lift_status := #LiftMoving;
           END_IF;*)

           IF (#Lift AND #Crane_status = #Stopped) THEN
               #Crane_QD.Lift := TRUE;
           ELSE
               #Crane_QD.Lift := FALSE;
           END_IF;

           IF ((#Setpoint <= #MAX_SETPOINT AND #Setpoint > 0)
               AND #Setpoint <> #Crane_target_position
               AND #Crane_status = #Stopped)
           THEN
               #Crane_target_position := #Setpoint;
               #Crane_status := #Moving;
           END_IF;

           #Check_forksL_move(IN := (#Forks_mLeft AND NOT #Forks_mRight AND NOT #Crane_IN.At_left),
                              PT := T#8s);

           #Check_forksR_move(IN := (#Forks_mRight AND NOT #Forks_mLeft AND NOT #Crane_IN.At_right),
                              PT := T#8s);

           #Check_forksM_move(IN := (NOT #Forks_mLeft AND NOT #Forks_mRight AND NOT #Crane_IN.At_middle),
                              PT := T#8s);

           (*
           #Check_lift_moving(IN:= (#Crane_status = #Stopped AND #Lift AND #Lift_status = #LiftMoving AND #Crane_IN.Moving_Z),
                              PT:=T#1s);

           #Check_lift_stuck(IN:=(#Lift_status = #LiftMoving),
                             PT:=T#8s);*)

           #Check_stacker_moving(IN:=(NOT(#Crane_IN.Moving_X OR #Crane_IN.Moving_Z)),
                                 PT:=T#2s); //#Crane_status = #Moving AND 

           #Check_stacker_stuck(IN := (#Crane_status = #Moving),
                                PT := T#25s);

           (*IF (#Check_lift_moving.Q) THEN
               #Lift_status := #LiftStopped;
           END_IF;

           IF (#Check_lift_stuck.Q) THEN
               #Lift_status := #LiftStopped; // PRELIMINARY OPERATION, MAY BE REPLACED IN FUTURE
                                             // ISSUE LIFT STUCK ALARM
           END_IF;*)

           IF (#Check_stacker_moving.Q) THEN
               #Crane_status := #Stopped;
           END_IF;

           IF (#Check_stacker_stuck.Q) THEN
               #Crane_status := #Stopped; //ISSUE ALARM STACKER CRANE STUCK
           END_IF;

           (*IF (#Check_forksL_move.Q) OR
              (#Check_forksM_move.Q) OR
              (#Check_forksR_move.Q)
           THEN
               #Crane_QD.Forks_left := FALSE; //ISSUE ALARM FORKS STUCK
               #Crane_QD.Forks_right := FALSE;
           END_IF;*)

       ELSIF (#Stop) THEN
           ;
       END_IF;
   END_IF;

   IF (#Reset) THEN
       #On_time.On_time_hours := 0;
       #On_time.On_time_mins := 0;
       #On_time.On_time_secs := 0;
       #Equipment_status := #Off;
   END_IF;

   IF (#Crane_QD.Forks_left OR
       #Crane_QD.Forks_right OR
       #Crane_QD.Lift OR
       #Crane_IN.Moving_X OR
       #Crane_IN.Moving_Z) THEN

       #Equipment_time_counter_Instance(Clock:=#Clock,
                                        On_time:=#On_time);

       #Equipment_status := #On;
   ELSE
       #Equipment_status := #Off;

   END_IF;
END_FUNCTION_BLOCK

FUNCTION "Reset_warehouse" : Void   // FC1, SCL
{ S7_Optimized_Access := 'TRUE' }
VERSION : 0.1
   VAR_IN_OUT
      Warehouse : Array[1..54] of Int;
   END_VAR
   VAR_TEMP
      Current_pos : Int;
   END_VAR
   VAR CONSTANT
      Capacity : Int := 54;
   END_VAR
BEGIN
   FOR #Current_pos := 1 TO #Capacity DO
       #Warehouse[#Current_pos] := 0;
   END_FOR;
END_FUNCTION

FUNCTION "Free_position" : Void   // FC2, SCL
{ S7_Optimized_Access := 'TRUE' }
VERSION : 0.1
   VAR_INPUT
      Warehouse : Array[1..54] of Int;
   END_VAR
   VAR_OUTPUT
      Free_position : Int;
      Free_shelves : Int;
      Occupied_shelves : Int;
   END_VAR
   VAR_TEMP
      Current_pos : Int;
   END_VAR
   VAR CONSTANT
      Capacity : Int := 54;
   END_VAR
BEGIN
   #Occupied_shelves := 0;

   FOR #Current_pos := 1 TO #Capacity DO
       IF(#Warehouse[#Current_pos] > 0) THEN
           #Occupied_shelves := #Occupied_shelves + 1;
       END_IF;
   END_FOR;

   #Free_shelves := #Capacity - #Occupied_shelves;

   FOR #Current_pos := 1 TO #Capacity DO
       IF (#Warehouse[#Current_pos] = 0) THEN
           #Free_position := #Current_pos;
           EXIT;
       END_IF;
   END_FOR;
END_FUNCTION

// folder: 03_Warehouse1

FUNCTION_BLOCK "Warehouse1_control"   // FB9, SCL
{ S7_Optimized_Access := 'TRUE' }
VERSION : 0.1
   VAR_INPUT
      Start : Bool;
      Stop : Bool;
      Reset : Bool;
      Mode : Bool;
      Clock : Bool;
      EntryCrane_IN : "Equip_crane_IN_t";
      ExitCrane_IN : "Equip_crane_IN_t";
      Entry_sensor : Bool;
   END_VAR
   VAR_OUTPUT
      EntryCrane_QD : "Equip_crane_QD_t";
      EntryCrane_TP : Int;
      ExitCrane_QD : "Equip_crane_QD_t";
      ExitCrane_TP : Int;
      WH1_load_conveyor : Bool;
   END_VAR
   VAR_IN_OUT
      Warehouse1 : Array[1..54] of Int;
      WH1_entry_crane_free : Bool;
   END_VAR
   VAR
      Entry_sensor_FB : "Sensor_control";
      Entry_crane_FB : "Crane_control";
      Exit_crane_FB : "Crane_control";
      WH1_load_conveyor_FB : "Conveyor_control";
      Entry_crane_SP : Int;
      Exit_crane_SP : Int;
      Entry_crane_state : Int;
      Exit_crane_state : Int;
      Entry_crane_lift : Bool;
      Entry_crane_fLeft : Bool;
      Entry_crane_fRight : Bool;
      Entry_crane_goto : Bool;
      Exit_crane_lift : Bool;
      Delay_forks_left_lift : TON_TIME;
      Pallet_lifted : TON_TIME;
      "Delay_forks_retract(redundant?)" : TON_TIME;
      Delay_entCrane_move_WH : TON_TIME;
      Pallet_lowered : TON_TIME;
      Delay_entCrane_move_HM : TON_TIME;
      Entry_sensor_free_delay : TON_TIME;
   END_VAR
   VAR CONSTANT
      MAN : Bool := 0;
      AUTO : Bool := 1;
      AtHome : Int := 0;
      PickupFromHome : Int := 1;
      GoToPlacePos : Int := 2;
      AtPlacePos : Int := 3;
      GotoHome : Int := 4;
      HOME_POS : Int := 55;
      WH_OCCUPIED : Int := 1;
      WH_EMPTY : Int := 0;
   END_VAR
BEGIN

   REGION FB_calls_for_equipment_and_sensors

       #Entry_crane_FB(Start:=#Start,
                       Stop:=#Stop,
                       Reset:=#Reset,
                       Mode:=#Mode,
                       Clock:=#Clock,
                       Forks_mLeft:=("HMI".MAN_CTRL.Warehouse1.Entry_crane.Forks_left)
                       OR (#Entry_crane_fLeft),
                       Forks_mRight:=("HMI".MAN_CTRL.Warehouse1.Entry_crane.Forks_right)
                       OR (#Entry_crane_fRight),
                       Lift:=("HMI".MAN_CTRL.Warehouse1.Entry_crane.Lift)
                       OR (#Entry_crane_lift),
                       Crane_IN:=#EntryCrane_IN,
                       Setpoint:=#Entry_crane_SP,
                       Crane_QD=>#EntryCrane_QD,
                       Crane_target_position=>#EntryCrane_TP);

       #Exit_crane_FB(Start:=#Start,
                      Stop:=#Stop,
                      Reset:=#Reset,
                      Mode:=#Mode,
                      Clock:=#Clock,
                      Forks_mLeft:=("HMI".MAN_CTRL.Warehouse1.Exit_crane.Forks_left),
                      Forks_mRight:=("HMI".MAN_CTRL.Warehouse1.Exit_crane.Forks_right),
                      Lift:=("HMI".MAN_CTRL.Warehouse1.Exit_crane.Lift),
                      Crane_IN:=#ExitCrane_IN,
                      Setpoint:=#Exit_crane_SP,
                      Crane_QD=>#ExitCrane_QD,
                      Crane_target_position=>#ExitCrane_TP);

       #WH1_load_conveyor_FB(Start:=#Start,
                             Stop:=#Stop,
                             Reset:=#Reset,
                             Mode:=#Mode,
                             Clock:=#Clock,
                             Fwd:=("HMI".MAN_CTRL.Warehouse1.WH1_load_conveyor)
                             OR (#WH1_entry_crane_free),
                             Bwd:=FALSE,
                             Conveyor_fwd=>#WH1_load_conveyor);

       #Entry_sensor_FB(Sensor:=#Entry_sensor,
                        Debounce_time:=T#100ms,
                        Timeout:=T#2000ms,
                        Enabled:=TRUE);

   END_REGION

   IF (#Reset) THEN
       "Reset_warehouse"(#Warehouse1);
       #Entry_crane_state := #GotoHome;
       #Exit_crane_state := #GotoHome;
       #Entry_crane_fLeft := FALSE;
       #Entry_crane_fRight := FALSE;
       #Entry_crane_lift := FALSE;
   END_IF;

   IF (#Mode = #AUTO) AND (#Start) THEN

       IF (#Entry_sensor_FB.Is_free) THEN
           #WH1_entry_crane_free := FALSE;
       END_IF;

       #Entry_sensor_free_delay(IN := #Entry_sensor_FB.Is_busy,
                                PT := T#2s);

       IF (#Entry_sensor_free_delay.Q) THEN
           #WH1_entry_crane_free := TRUE;
       END_IF;

       #EntryCrane_TP := #Entry_crane_SP;

       REGION Entry_crane_state_machine
           CASE #Entry_crane_state OF
               #AtHome:
                   #Entry_crane_lift := FALSE;
                   #Entry_crane_fLeft := FALSE;
                   #Entry_crane_fRight := FALSE;

                   IF (NOT #WH1_entry_crane_free AND NOT(#EntryCrane_IN.Moving_X AND #EntryCrane_IN.Moving_Z)) THEN
                       #Entry_crane_state := #PickupFromHome; 
                   END_IF;

               #PickupFromHome:
                   IF (#EntryCrane_IN.At_middle) THEN
                       #Entry_crane_fLeft := TRUE;
                       #Entry_crane_fRight := FALSE;
                   END_IF;

                   IF (#EntryCrane_IN.At_left) THEN
                       #Entry_crane_lift := TRUE;
                   END_IF;

                   #Pallet_lifted(IN:=#Entry_crane_lift,
                                  PT:=T#2s);

                   IF (#Pallet_lifted.Q) THEN
                       #Entry_crane_fLeft := FALSE;
                   END_IF;

                   IF (#EntryCrane_IN.At_middle AND NOT #Entry_crane_fLeft) THEN
                       #Entry_crane_state := #GoToPlacePos;
                   END_IF;

               #GoToPlacePos:
                   IF (#EntryCrane_IN.At_middle) THEN
                       #Entry_crane_goto := TRUE;
                       "Free_position"(Warehouse := #Warehouse1,
                                       "Free_position" => #Entry_crane_SP,
                                       Free_shelves => "Warehouse1".Free_positions,
                                       Occupied_shelves => "Warehouse1".Occupied_positions);
                   END_IF;

                   IF (#Delay_entCrane_move_WH.Q) THEN
                       #Entry_crane_state := #AtPlacePos;
                       #Entry_crane_goto := FALSE;
                   END_IF;

                   #Delay_entCrane_move_WH(IN:= #Entry_crane_goto AND NOT (#EntryCrane_IN.Moving_X AND #EntryCrane_IN.Moving_Z),
                                           PT:=T#2s);

               #AtPlacePos:
                   IF (#EntryCrane_IN.At_middle AND #Entry_crane_lift) THEN
                       #Entry_crane_fRight := TRUE;
                       #Entry_crane_fLeft := FALSE;
                   END_IF;

                   IF (#EntryCrane_IN.At_right) THEN
                       #Entry_crane_lift := FALSE;
                   END_IF;

                   #Pallet_lowered(IN:=(NOT #Entry_crane_lift),
                                       PT:=T#2s);

                   IF (#Pallet_lowered.Q) THEN
                       #Entry_crane_fRight := FALSE;
                       #Warehouse1[#Entry_crane_SP] := #WH_OCCUPIED;
                   END_IF;

                   IF (#EntryCrane_IN.At_middle AND NOT (#Entry_crane_fRight)) THEN
                       #Entry_crane_state := #GotoHome;
                   END_IF;

               #GotoHome:
                   IF (#EntryCrane_IN.At_middle) THEN
                       #Entry_crane_goto := TRUE;
                       #Entry_crane_SP := #HOME_POS;
                   END_IF;

                   IF (#Delay_entCrane_move_HM.Q) THEN
                       #Entry_crane_state := #AtHome;
                       #Entry_crane_goto := FALSE;
                   END_IF;

                   #Delay_entCrane_move_HM(IN:=#Entry_crane_goto AND NOT (#EntryCrane_IN.Moving_X AND #EntryCrane_IN.Moving_Z),
                                           PT:=T#2s);

               ELSE 
                   ;
           END_CASE;
       END_REGION 

       REGION Exit_crane_state_machine
           CASE #Exit_crane_state OF
               #AtHome:
                   ;
               2:  
                   ;
               ELSE  
                   ;
           END_CASE;
       END_REGION

   END_IF;
END_FUNCTION_BLOCK

// folder: 04_Gantry1_palletizer

FUNCTION_BLOCK "Gantry1_Palletizer"   // FB7, SCL
{ S7_Optimized_Access := 'TRUE' }
VERSION : 0.1
BEGIN
END_FUNCTION_BLOCK

// folder: 05_Elevator_control

FUNCTION_BLOCK "Elevator_control"   // FB3, SCL
{ S7_Optimized_Access := 'TRUE' }
VERSION : 0.1
   VAR_INPUT
      Start : Bool;
      Stop : Bool;
      Reset : Bool;
      Mode : Bool;
      Clock : Bool;
      Elevator_IN : "Equip_elevator_IN_t";
      Setpoint : Real;
   END_VAR
   VAR_OUTPUT
      Elevator_QD : "Equip_elevator_QD_t";
      Elevator_QW : "Equip_elevator_QW_t";
   END_VAR
   VAR
      On_time : "Info_OnTime_t";
      Equipment_time_counter_Instance : "Equipment_time_counter";
      Status : Int;
   END_VAR
   VAR CONSTANT
      MAN : Bool := 0;
      AUTO : Bool := 1;
      On : Int := 0;
      Off : Int := 1;
   END_VAR
BEGIN
   IF (#Mode = #MAN) THEN
       "Manual_control"();
   END_IF;

   IF (#Mode = #AUTO) THEN
       IF (#Start) THEN
           ;
       ELSIF (#Stop) THEN
           ;
       END_IF;
   END_IF;

   IF (#Reset) THEN
       #On_time.On_time_hours := 0;
       #On_time.On_time_mins := 0;
       #On_time.On_time_secs := 0;
       #Status := #Off;
   END_IF;

   IF (#Elevator_QD.Conveyor_fwd OR
       #Elevator_QD.Conveyor_bwd)
   THEN

       #Equipment_time_counter_Instance(Clock:=#Clock,
                                        On_time:=#On_time);


       #Status := #On;
   ELSE
       #Status := #Off;

   END_IF;
END_FUNCTION_BLOCK

// folder: General_functions

FUNCTION_BLOCK "Equipment_time_counter"   // FB6, SCL
{ S7_Optimized_Access := 'TRUE' }
VERSION : 0.1
   VAR_INPUT
      Clock : Bool;
   END_VAR
   VAR_IN_OUT
      On_time : "Info_OnTime_t";
   END_VAR
   VAR RETAIN
      IEC_TimeCounterSECS_Instance : CTU_INT;
      IEC_TimeCounterMINS_Instance : CTU_INT;
      IEC_TimeCounterHOURS_Instance : CTU_INT;
   END_VAR
BEGIN
   #IEC_TimeCounterSECS_Instance(CU := #Clock,
                                 R := FALSE,
                                 PV := 60,
                                 CV => #On_time.On_time_secs);

   IF (#IEC_TimeCounterSECS_Instance.CV = 60) THEN
       #IEC_TimeCounterMINS_Instance(CU := 1,
                                     R := FALSE,
                                     PV := 60,
                                     CV => #On_time.On_time_mins);
       #On_time.On_time_secs := 0;
   END_IF;

   IF (#IEC_TimeCounterMINS_Instance.CV = 60) THEN

       #IEC_TimeCounterHOURS_Instance(CU := 1,
                                      R := FALSE,
                                      PV := 2000,
                                      CV => #On_time.On_time_hours);
       #On_time.On_time_mins := 0;
   END_IF;

   // Switch to this:
   // On_time.On_time_ms := On_time.On_time_ms + OB1_PREV_CYCLE;
END_FUNCTION_BLOCK

FUNCTION_BLOCK "Sensor_control"   // FB10, SCL
{ S7_Optimized_Access := 'TRUE' }
VERSION : 0.1
   VAR_INPUT
      Sensor : Bool;
      Debounce_time : Time;
      Timeout : Time;
      Enabled : Bool;
   END_VAR
   VAR_OUTPUT
      Is_free : Bool;
      Is_busy : Bool;
      R_edge : Bool;
      F_edge : Bool;
      Flickering : Bool;
      Raw_signal : Bool;
   END_VAR
   VAR
      Debouncing_ON : TON_TIME;
      Debouncing_OFF : TOF_TIME;
      R_TRIG_Instance : R_TRIG;
      F_TRIG_Instance : F_TRIG;
      Timer_flickering : TON_TIME;
   END_VAR
BEGIN
   IF (#Enabled) THEN
       #Raw_signal := #Sensor;

       #Debouncing_ON(IN:=#Sensor,
                      PT:=#Debounce_time);


       #Is_busy := #Debouncing_ON.Q;

       #Debouncing_OFF(IN:= (NOT #Sensor),
                       PT:=#Debounce_time);


       #Is_free := #Debouncing_OFF.Q;

       #R_TRIG_Instance(CLK:=#Debouncing_ON.Q);

       #R_edge := #R_TRIG_Instance.Q;

       #F_TRIG_Instance(CLK:=#Debouncing_OFF.Q);

       #F_edge := #F_TRIG_Instance.Q;

       #Timer_flickering(IN:=(NOT #Is_busy AND NOT #Is_free),
                         PT:=#Timeout,
                         Q=>#Flickering);

   END_IF;
END_FUNCTION_BLOCK

FUNCTION "Norm_and_scale" : Void   // FC5, LAD
{ S7_Optimized_Access := 'TRUE' }
VERSION : 0.1
   VAR_INPUT
      Input : Int;
      Norm_min : Int;
      Norm_max : Int;
      Scale_min : Int;
      Scale_max : Int;
   END_VAR
   VAR_OUTPUT
      Output : Real;
   END_VAR
   VAR_TEMP
      Temp : Real;
   END_VAR
BEGIN

REGION Network 1: Norm and scale input
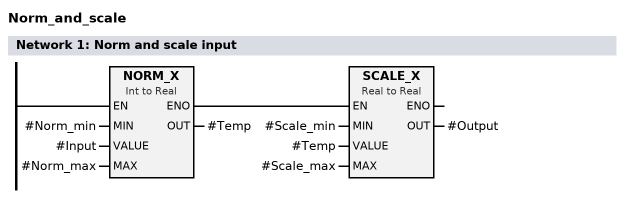
   RUNG wire#powerrail
      { S7_Templates := "[SrcType := Int, DestType := Real]" } Normalize(min := #Norm_min, value := #Input, max := #Norm_max, out => #Temp)
      { S7_Templates := "[SrcType := Real, DestType := Real]" } Scale(min := #Scale_min, value := #Temp, max := #Scale_max, out => #Output)
   END_RUNG
   // the same network as SCL:
   #Temp := NORM_X(MIN := #Norm_min, VALUE := #Input, MAX := #Norm_max);
   #Output := SCALE_X(MIN := #Scale_min, VALUE := #Temp, MAX := #Scale_max);
END_REGION
END_FUNCTION

(* ===== HMI "HMI_RT_1" =====

ScreenModuleEditorView "Faceplate_Pallet2" 640x480
   SymbolLibrary "Symbol library_3" at 10,67 size 186x48
   SymbolLibrary "Symbol library_1" at 36,10 size 76x65
   SymbolLibrary "Symbol library_2" at 95,10 size 73x65
*)

(* ===== HMI "HMI_RT_1" =====

ScreenModuleEditorView "Faceplate_Pallet2" 640x480
   SymbolLibrary "Symbol library_3" at 10,67 size 186x48
   SymbolLibrary "Symbol library_1" at 36,10 size 76x65
   SymbolLibrary "Symbol library_2" at 95,10 size 73x65
*)

(* ===== HMI "HMI_RT_1" =====
system functions are stored by id; their names below are inferred from use
connection "HMI_Connection_1": ETHERNET, S7_1200_OMS

HMI tags "Default tag table"
   "Tag_ScreenNumber" : UInt, internal

screen "Root screen" 800x420, template "Template_1"
   on GenerateScreen: SetTag("Tag_ScreenNumber", 1)
*)